SUBAPPLICATION GreenRedBackground3 (* Hintergrundfarbe (TRUE -> Rot, FALSE -> Grün) für 3 Objekte *)
  (* Standard: 61499-2 *)
  (* Version 1.0, 2022-11-10, franz *)
  PACKAGE MyLib::sys;
  IMPORT isobus::UT::Q::const::colours;
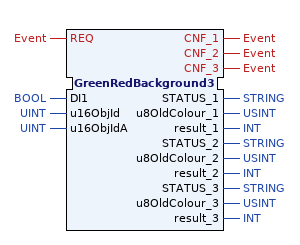
  EVENT_INPUT
    REQ; (* Normal Execution Request *)
  END_EVENT
  EVENT_OUTPUT
    CNF_1; (* Execution Confirmation *)
    CNF_2;
    CNF_3;
  END_EVENT
  VAR_INPUT
    DI1 : BOOL; (* Selector *)
    u16ObjId : UINT; (* Object ID Softkey *)
    u16ObjIdA : UINT; (* Object ID AUX *)
  END_VAR
  VAR_OUTPUT
    STATUS_1 : STRING; (* Service Status *)
    u8OldColour_1 : USINT; (* Old value of ID *)
    result_1 : INT; (* retval see description *)
    STATUS_2 : STRING; (* Service Status *)
    u8OldColour_2 : USINT; (* Old value of ID *)
    result_2 : INT; (* retval see description *)
    STATUS_3 : STRING; (* Service Status *)
    u8OldColour_3 : USINT; (* Old value of ID *)
    result_3 : INT; (* retval see description *)
  END_VAR
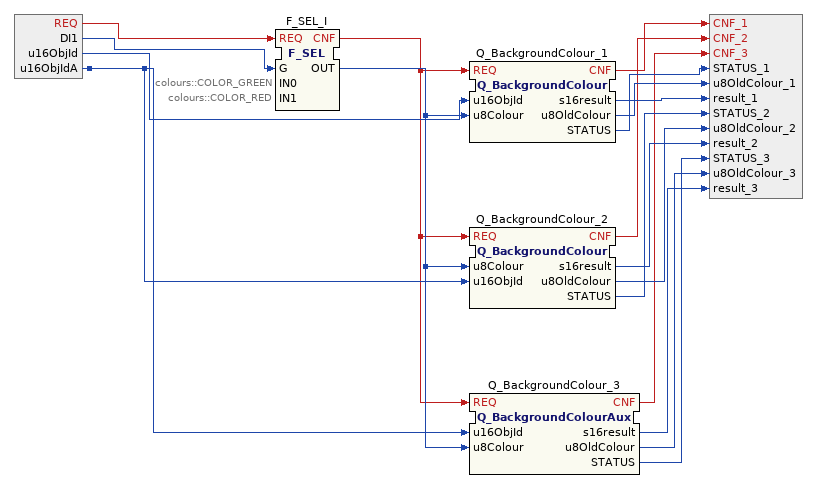
  FBS
    Q_BackgroundColour_1 : isobus::UT::Q::Q_BackgroundColour;
    Q_BackgroundColour_2 : isobus::UT::Q::Q_BackgroundColour;
    Q_BackgroundColour_3 : isobus::UT::Q::Q_BackgroundColourAux;
    F_SEL_I : iec61131::selection::F_SEL(IN0 := colours::COLOR_GREEN, IN1 := colours::COLOR_RED);
  END_FBS
  EVENT_CONNECTIONS
    Q_BackgroundColour_3.CNF TO CNF_3;
    Q_BackgroundColour_2.CNF TO CNF_2;
    Q_BackgroundColour_1.CNF TO CNF_1;
    REQ TO F_SEL_I.REQ;
    F_SEL_I.CNF TO Q_BackgroundColour_1.REQ;
    F_SEL_I.CNF TO Q_BackgroundColour_2.REQ;
    F_SEL_I.CNF TO Q_BackgroundColour_3.REQ;
  END_CONNECTIONS
  DATA_CONNECTIONS
    u16ObjId TO Q_BackgroundColour_1.u16ObjId;
    u16ObjIdA TO Q_BackgroundColour_3.u16ObjId;
    Q_BackgroundColour_3.s16result TO result_3;
    Q_BackgroundColour_3.u8OldColour TO u8OldColour_3;
    Q_BackgroundColour_3.STATUS TO STATUS_3;
    Q_BackgroundColour_2.s16result TO result_2;
    Q_BackgroundColour_2.u8OldColour TO u8OldColour_2;
    Q_BackgroundColour_2.STATUS TO STATUS_2;
    Q_BackgroundColour_1.s16result TO result_1;
    Q_BackgroundColour_1.u8OldColour TO u8OldColour_1;
    Q_BackgroundColour_1.STATUS TO STATUS_1;
    DI1 TO F_SEL_I.G;
    F_SEL_I.OUT TO Q_BackgroundColour_1.u8Colour;
    F_SEL_I.OUT TO Q_BackgroundColour_2.u8Colour;
    F_SEL_I.OUT TO Q_BackgroundColour_3.u8Colour;
    u16ObjIdA TO Q_BackgroundColour_2.u16ObjId;
  END_CONNECTIONS
END_SUBAPPLICATION
